{attribute addProperty BoxType "EK1122-0000-0018"}
{attribute addProperty Id "Beckhoff_EK15xxsub_EK1100EK1100_179A0949162A_0001_EK1501_0000_0016EK1501_963BF4D7344.25A_0002_EK1501_0000_0017EK1501_963BF4D7344.25A_0003_EK1501_0000_0018EK1501_963BF4D7344.25A_0004_EK1501_0000_0019EK1501_963BF4D7344.25A_0005_EK1501_0010_0016EK1501_963BF4D7344.25A_0006_EK1501_0010_0017EK1501_963BF4D7344.25A_0007_EK1501_0010_0018EK1501_963BF4D7344.25A_0008_EK1501_0100_0016EK1501_963BF4D7344.25A_0020_EK1541_0000_0016EK1541_963BF4D7344.25A_0021_EK1541_0000_0017EK1541_963BF4D7344.25A_0022_EK1541_0000_0018EK1541_963BF4D7344.25"}
{attribute addProperty CRC "4102180946"}
{attribute addProperty SizeInBites "390"}
{attribute addProperty SizeInBytes "48.75"}
TYPE Beckhoff_EK15xxEK1122_F4825052 EXTENDS EK1122_179A0949 :
STRUCT
	{attribute addProperty Name "Beckhoff_EK15xxsub_EK1100"}
	Beckhoff_EK15xxsub_EK1100 : EK1100_179A0949;
	{attribute addProperty Name "A_0001_EK1501_0000_0016"}
	A_0001_EK1501_0000_0016 : EK1501_963BF4D7;
	{attribute addProperty Name "A_0002_EK1501_0000_0017"}
	A_0002_EK1501_0000_0017 : EK1501_963BF4D7;
	{attribute addProperty Name "A_0003_EK1501_0000_0018"}
	A_0003_EK1501_0000_0018 : EK1501_963BF4D7;
	{attribute addProperty Name "A_0004_EK1501_0000_0019"}
	A_0004_EK1501_0000_0019 : EK1501_963BF4D7;
	{attribute addProperty Name "A_0005_EK1501_0010_0016"}
	A_0005_EK1501_0010_0016 : EK1501_963BF4D7;
	{attribute addProperty Name "A_0006_EK1501_0010_0017"}
	A_0006_EK1501_0010_0017 : EK1501_963BF4D7;
	{attribute addProperty Name "A_0007_EK1501_0010_0018"}
	A_0007_EK1501_0010_0018 : EK1501_963BF4D7;
	{attribute addProperty Name "A_0008_EK1501_0100_0016"}
	A_0008_EK1501_0100_0016 : EK1501_963BF4D7;
	{attribute addProperty Name "A_0020_EK1541_0000_0016"}
	A_0020_EK1541_0000_0016 : EK1541_963BF4D7;
	{attribute addProperty Name "A_0021_EK1541_0000_0017"}
	A_0021_EK1541_0000_0017 : EK1541_963BF4D7;
	{attribute addProperty Name "A_0022_EK1541_0000_0018"}
	A_0022_EK1541_0000_0018 : EK1541_963BF4D7;
END_STRUCT
END_TYPE

(* stored: Version 1.2.0.0, ProductVersion 3.1.4024.9
   DUT Beckhoff_EK15xxEK1122_F4825052: Id {68642fc9-b8b8-417e-98a0-5f0aa12c9b52} *)
